(* Visualisation PLC_VISU
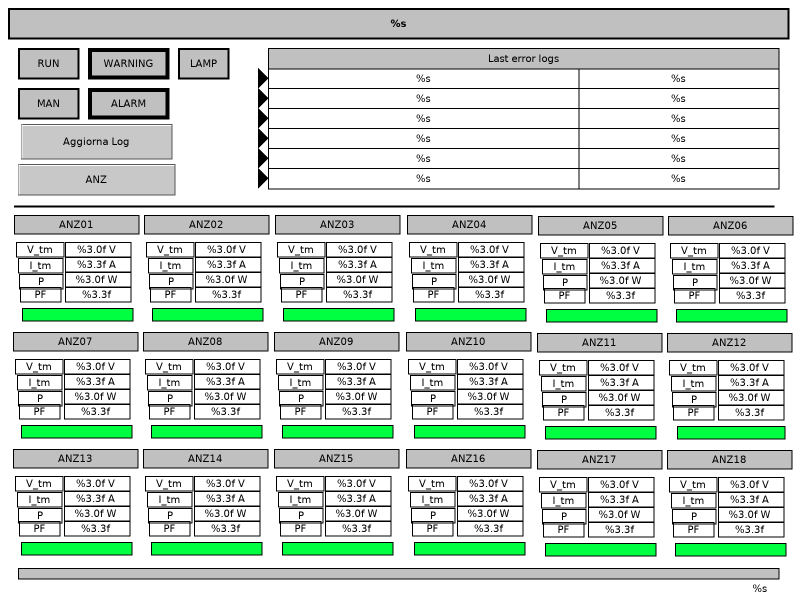
rectangle at (10,10)-(791,41): text "%s"; shows .Plant_NAME
rectangle at (530,580)-(771,601): text "%s"; shows Sys.Time_LogString
rounded rectangle at (20,50)-(81,81): text "RUN"; alarm colour if NOT Mode_Manual; runs INTERN ASSIGN Mode_Manual:=(FALSE)
rounded rectangle at (20,90)-(81,121): text "MAN"; alarm colour if Mode_Manual; runs INTERN ASSIGN Mode_Manual:=(TRUE)
rectangle at (580,70)-(781,91): text "%s"; shows Sys.LastLogs_Msg[0]
polygon at (260,170)-(270,190): invisible if Sys.LastLogs_Idx<>0
rectangle at (580,90)-(781,111): text "%s"; shows Sys.LastLogs_Msg[1]
polygon at (260,70)-(270,90): invisible if Sys.LastLogs_Idx<>1
rectangle at (580,110)-(781,131): text "%s"; shows Sys.LastLogs_Msg[2]
polygon at (260,90)-(270,110): invisible if Sys.LastLogs_Idx<>2
rectangle at (580,130)-(781,151): text "%s"; shows Sys.LastLogs_Msg[3]
polygon at (260,110)-(270,130): invisible if Sys.LastLogs_Idx<>3
rectangle at (580,150)-(781,171): text "%s"; shows Sys.LastLogs_Msg[4]
polygon at (260,130)-(270,150): invisible if Sys.LastLogs_Idx<>4
rectangle at (580,170)-(781,191): text "%s"; shows Sys.LastLogs_Msg[5]
polygon at (260,150)-(270,170): invisible if Sys.LastLogs_Idx<>5
rectangle at (270,70)-(581,91): text "%s"; shows Sys.LastLogs_Dat[0]
rectangle at (270,90)-(581,111): text "%s"; shows Sys.LastLogs_Dat[1]
rectangle at (270,110)-(581,131): text "%s"; shows Sys.LastLogs_Dat[2]
rectangle at (270,130)-(581,151): text "%s"; shows Sys.LastLogs_Dat[3]
rectangle at (270,150)-(581,171): text "%s"; shows Sys.LastLogs_Dat[4]
rectangle at (270,170)-(581,191): text "%s"; shows Sys.LastLogs_Dat[5]
rectangle at (90,90)-(171,121): text "ALARM"; alarm colour if Sys.Alarm; runs INTERN ASSIGN Mode_Manual:=(FALSE)
rectangle at (90,50)-(171,81): text "WARNING"; alarm colour if Sys.Warning; runs INTERN ASSIGN Mode_Manual:=(TRUE)
rectangle at (270,50)-(781,71): text "Last error logs"
rounded rectangle at (180,50)-(231,81): text "LAMP"; alarm colour if LAMP_AL
button at (23,126)-(174,161): text "Aggiorna Log"; taps PLC_PRG.HMI_AggiornaLog
button at (20,166)-(177,197): text "ANZ"; opens VIS_ANZ
rectangle at (67,244)-(133,259): text "%3.0f V"; shows .ANZ01.Voltage_L1_L2
rectangle at (18,244)-(66,259): text "V_tm"
rectangle at (20,260)-(65,275): text "I_tm"
rectangle at (21,276)-(65,291): text "P"
rectangle at (22,289)-(63,304): text "PF"
rectangle at (67,259)-(133,274): text "%3.3f A"; shows .ANZ01.Current_L1
rectangle at (67,274)-(133,289): text "%3.0f W"; shows .ANZ01.ActivePower
rectangle at (67,289)-(133,304): text "%3.3f"; shows .ANZ01.Power_factor_L1
rectangle at (24,310)-(135,323): alarm colour if .ANZ01.AllarmeNodo
rectangle at (16,217)-(141,236): text "ANZ01"
rectangle at (197,244)-(263,259): text "%3.0f V"; shows .ANZ02.Voltage_L1_L2
rectangle at (148,244)-(196,259): text "V_tm"
rectangle at (150,260)-(195,275): text "I_tm"
rectangle at (151,276)-(195,291): text "P"
rectangle at (152,289)-(193,304): text "PF"
rectangle at (197,259)-(263,274): text "%3.3f A"; shows .ANZ02.Current_L1
rectangle at (197,274)-(263,289): text "%3.0f W"; shows .ANZ02.ActivePower
rectangle at (197,289)-(263,304): text "%3.3f"; shows .ANZ02.Power_factor_L1
rectangle at (154,310)-(265,323): alarm colour if .ANZ02.AllarmeNodo
rectangle at (146,217)-(271,236): text "ANZ02"
rectangle at (328,244)-(394,259): text "%3.0f V"; shows .ANZ03.Voltage_L1_L2
rectangle at (279,244)-(327,259): text "V_tm"
rectangle at (281,260)-(326,275): text "I_tm"
rectangle at (282,276)-(326,291): text "P"
rectangle at (283,289)-(324,304): text "PF"
rectangle at (328,259)-(394,274): text "%3.3f A"; shows .ANZ03.Current_L1
rectangle at (328,274)-(394,289): text "%3.0f W"; shows .ANZ03.ActivePower
rectangle at (328,289)-(394,304): text "%3.3f"; shows .ANZ03.Power_factor_L1
rectangle at (285,310)-(396,323): alarm colour if .ANZ03.AllarmeNodo
rectangle at (277,217)-(402,236): text "ANZ03"
rectangle at (460,244)-(526,259): text "%3.0f V"; shows .ANZ04.Voltage_L1_L2
rectangle at (411,244)-(459,259): text "V_tm"
rectangle at (413,260)-(458,275): text "I_tm"
rectangle at (414,276)-(458,291): text "P"
rectangle at (415,289)-(456,304): text "PF"
rectangle at (460,259)-(526,274): text "%3.3f A"; shows .ANZ04.Current_L1
rectangle at (460,274)-(526,289): text "%3.0f W"; shows .ANZ04.ActivePower
rectangle at (460,289)-(526,304): text "%3.3f"; shows .ANZ04.Power_factor_L1
rectangle at (417,310)-(528,323): alarm colour if .ANZ04.AllarmeNodo
rectangle at (409,217)-(534,236): text "ANZ04"
rectangle at (591,245)-(657,260): text "%3.0f V"; shows .ANZ05.Voltage_L1_L2
rectangle at (542,245)-(590,260): text "V_tm"
rectangle at (544,261)-(589,276): text "I_tm"
rectangle at (545,277)-(589,292): text "P"
rectangle at (546,290)-(587,305): text "PF"
rectangle at (591,260)-(657,275): text "%3.3f A"; shows .ANZ05.Current_L1
rectangle at (591,275)-(657,290): text "%3.0f W"; shows .ANZ05.ActivePower
rectangle at (591,290)-(657,305): text "%3.3f"; shows .ANZ05.Power_factor_L1
rectangle at (548,311)-(659,324): alarm colour if .ANZ05.AllarmeNodo
rectangle at (540,218)-(665,237): text "ANZ05"
rectangle at (721,245)-(787,260): text "%3.0f V"; shows .ANZ06.Voltage_L1_L2
rectangle at (672,245)-(720,260): text "V_tm"
rectangle at (674,261)-(719,276): text "I_tm"
rectangle at (675,277)-(719,292): text "P"
rectangle at (676,290)-(717,305): text "PF"
rectangle at (721,260)-(787,275): text "%3.3f A"; shows .ANZ06.Current_L1
rectangle at (721,275)-(787,290): text "%3.0f W"; shows .ANZ06.ActivePower
rectangle at (721,290)-(787,305): text "%3.3f"; shows .ANZ06.Power_factor_L1
rectangle at (678,311)-(789,324): alarm colour if .ANZ06.AllarmeNodo
rectangle at (670,218)-(795,237): text "ANZ06"
rectangle at (66,361)-(132,376): text "%3.0f V"; shows .ANZ07.Voltage_L1_L2
rectangle at (17,361)-(65,376): text "V_tm"
rectangle at (19,377)-(64,392): text "I_tm"
rectangle at (20,393)-(64,408): text "P"
rectangle at (21,406)-(62,421): text "PF"
rectangle at (66,376)-(132,391): text "%3.3f A"; shows .ANZ07.Current_L1
rectangle at (66,391)-(132,406): text "%3.0f W"; shows .ANZ07.ActivePower
rectangle at (66,406)-(132,421): text "%3.3f"; shows .ANZ07.Power_factor_L1
rectangle at (23,427)-(134,440): alarm colour if .ANZ07.AllarmeNodo
rectangle at (15,334)-(140,353): text "ANZ07"
rectangle at (196,361)-(262,376): text "%3.0f V"; shows .ANZ08.Voltage_L1_L2
rectangle at (147,361)-(195,376): text "V_tm"
rectangle at (149,377)-(194,392): text "I_tm"
rectangle at (150,393)-(194,408): text "P"
rectangle at (151,406)-(192,421): text "PF"
rectangle at (196,376)-(262,391): text "%3.3f A"; shows .ANZ08.Current_L1
rectangle at (196,391)-(262,406): text "%3.0f W"; shows .ANZ08.ActivePower
rectangle at (196,406)-(262,421): text "%3.3f"; shows .ANZ08.Power_factor_L1
rectangle at (153,427)-(264,440): alarm colour if .ANZ08.AllarmeNodo
rectangle at (145,334)-(270,353): text "ANZ08"
rectangle at (327,361)-(393,376): text "%3.0f V"; shows .ANZ09.Voltage_L1_L2
rectangle at (278,361)-(326,376): text "V_tm"
rectangle at (280,377)-(325,392): text "I_tm"
rectangle at (281,393)-(325,408): text "P"
rectangle at (282,406)-(323,421): text "PF"
rectangle at (327,376)-(393,391): text "%3.3f A"; shows .ANZ09.Current_L1
rectangle at (327,391)-(393,406): text "%3.0f W"; shows .ANZ09.ActivePower
rectangle at (327,406)-(393,421): text "%3.3f"; shows .ANZ09.Power_factor_L1
rectangle at (284,427)-(395,440): alarm colour if .ANZ09.AllarmeNodo
rectangle at (276,334)-(401,353): text "ANZ09"
rectangle at (459,361)-(525,376): text "%3.0f V"; shows .ANZ10.Voltage_L1_L2
rectangle at (410,361)-(458,376): text "V_tm"
rectangle at (412,377)-(457,392): text "I_tm"
rectangle at (413,393)-(457,408): text "P"
rectangle at (414,406)-(455,421): text "PF"
rectangle at (459,376)-(525,391): text "%3.3f A"; shows .ANZ10.Current_L1
rectangle at (459,391)-(525,406): text "%3.0f W"; shows .ANZ10.ActivePower
rectangle at (459,406)-(525,421): text "%3.3f"; shows .ANZ10.Power_factor_L1
rectangle at (416,427)-(527,440): alarm colour if .ANZ10.AllarmeNodo
rectangle at (408,334)-(533,353): text "ANZ10"
rectangle at (590,362)-(656,377): text "%3.0f V"; shows .ANZ11.Voltage_L1_L2
rectangle at (541,362)-(589,377): text "V_tm"
rectangle at (543,378)-(588,393): text "I_tm"
rectangle at (544,394)-(588,409): text "P"
rectangle at (545,407)-(586,422): text "PF"
rectangle at (590,377)-(656,392): text "%3.3f A"; shows .ANZ11.Current_L1
rectangle at (590,392)-(656,407): text "%3.0f W"; shows .ANZ11.ActivePower
rectangle at (590,407)-(656,422): text "%3.3f"; shows .ANZ11.Power_factor_L1
rectangle at (547,428)-(658,441): alarm colour if .ANZ11.AllarmeNodo
rectangle at (539,335)-(664,354): text "ANZ11"
rectangle at (720,362)-(786,377): text "%3.0f V"; shows .ANZ12.Voltage_L1_L2
rectangle at (671,362)-(719,377): text "V_tm"
rectangle at (673,378)-(718,393): text "I_tm"
rectangle at (674,394)-(718,409): text "P"
rectangle at (675,407)-(716,422): text "PF"
rectangle at (720,377)-(786,392): text "%3.3f A"; shows .ANZ12.Current_L1
rectangle at (720,392)-(786,407): text "%3.0f W"; shows .ANZ12.ActivePower
rectangle at (720,407)-(786,422): text "%3.3f"; shows .ANZ12.Power_factor_L1
rectangle at (669,335)-(794,354): text "ANZ12"
rectangle at (66,478)-(132,493): text "%3.0f V"; shows .ANZ13.Voltage_L1_L2
rectangle at (17,478)-(65,493): text "V_tm"
rectangle at (19,494)-(64,509): text "I_tm"
rectangle at (20,510)-(64,525): text "P"
rectangle at (21,523)-(62,538): text "PF"
rectangle at (66,493)-(132,508): text "%3.3f A"; shows .ANZ13.Current_L1
rectangle at (66,508)-(132,523): text "%3.0f W"; shows .ANZ13.ActivePower
rectangle at (66,523)-(132,538): text "%3.3f"; shows .ANZ13.Power_factor_L1
rectangle at (23,544)-(134,557): alarm colour if .ANZ13.AllarmeNodo
rectangle at (15,451)-(140,470): text "ANZ13"
rectangle at (196,478)-(262,493): text "%3.0f V"; shows .ANZ14.Voltage_L1_L2
rectangle at (147,478)-(195,493): text "V_tm"
rectangle at (149,494)-(194,509): text "I_tm"
rectangle at (150,510)-(194,525): text "P"
rectangle at (151,523)-(192,538): text "PF"
rectangle at (196,493)-(262,508): text "%3.3f A"; shows .ANZ14.Current_L1
rectangle at (196,508)-(262,523): text "%3.0f W"; shows .ANZ14.ActivePower
rectangle at (196,523)-(262,538): text "%3.3f"; shows .ANZ14.Power_factor_L1
rectangle at (153,544)-(264,557): alarm colour if .ANZ14.AllarmeNodo
rectangle at (145,451)-(270,470): text "ANZ14"
rectangle at (327,478)-(393,493): text "%3.0f V"; shows .ANZ15.Voltage_L1_L2
rectangle at (278,478)-(326,493): text "V_tm"
rectangle at (280,494)-(325,509): text "I_tm"
rectangle at (281,510)-(325,525): text "P"
rectangle at (282,523)-(323,538): text "PF"
rectangle at (327,493)-(393,508): text "%3.3f A"; shows .ANZ15.Current_L1
rectangle at (327,508)-(393,523): text "%3.0f W"; shows .ANZ15.ActivePower
rectangle at (327,523)-(393,538): text "%3.3f"; shows .ANZ15.Power_factor_L1
rectangle at (284,544)-(395,557): alarm colour if .ANZ15.AllarmeNodo
rectangle at (276,451)-(401,470): text "ANZ15"
rectangle at (459,478)-(525,493): text "%3.0f V"; shows .ANZ16.Voltage_L1_L2
rectangle at (410,478)-(458,493): text "V_tm"
rectangle at (412,494)-(457,509): text "I_tm"
rectangle at (413,510)-(457,525): text "P"
rectangle at (414,523)-(455,538): text "PF"
rectangle at (459,493)-(525,508): text "%3.3f A"; shows .ANZ16.Current_L1
rectangle at (459,508)-(525,523): text "%3.0f W"; shows .ANZ16.ActivePower
rectangle at (459,523)-(525,538): text "%3.3f"; shows .ANZ16.Power_factor_L1
rectangle at (416,544)-(527,557): alarm colour if .ANZ16.AllarmeNodo
rectangle at (408,451)-(533,470): text "ANZ16"
rectangle at (590,479)-(656,494): text "%3.0f V"; shows .ANZ17.Voltage_L1_L2
rectangle at (541,479)-(589,494): text "V_tm"
rectangle at (543,495)-(588,510): text "I_tm"
rectangle at (544,511)-(588,526): text "P"
rectangle at (545,524)-(586,539): text "PF"
rectangle at (590,494)-(656,509): text "%3.3f A"; shows .ANZ17.Current_L1
rectangle at (590,509)-(656,524): text "%3.0f W"; shows .ANZ17.ActivePower
rectangle at (590,524)-(656,539): text "%3.3f"; shows .ANZ17.Power_factor_L1
rectangle at (547,545)-(658,558): alarm colour if .ANZ17.AllarmeNodo
rectangle at (539,452)-(664,471): text "ANZ17"
rectangle at (720,479)-(786,494): text "%3.0f V"; shows .ANZ18.Voltage_L1_L2
rectangle at (671,479)-(719,494): text "V_tm"
rectangle at (673,495)-(718,510): text "I_tm"
rectangle at (674,511)-(718,526): text "P"
rectangle at (675,524)-(716,539): text "PF"
rectangle at (720,494)-(786,509): text "%3.3f A"; shows .ANZ18.Current_L1
rectangle at (720,509)-(786,524): text "%3.0f W"; shows .ANZ18.ActivePower
rectangle at (720,524)-(786,539): text "%3.3f"; shows .ANZ18.Power_factor_L1
rectangle at (677,545)-(788,558): alarm colour if .ANZ18.AllarmeNodo
rectangle at (669,452)-(794,471): text "ANZ18"
rectangle at (679,428)-(787,441): alarm colour if .ANZ12.AllarmeNodo
20 more shapes without text or variables
*)

(* Visualisation VIS_ANZ
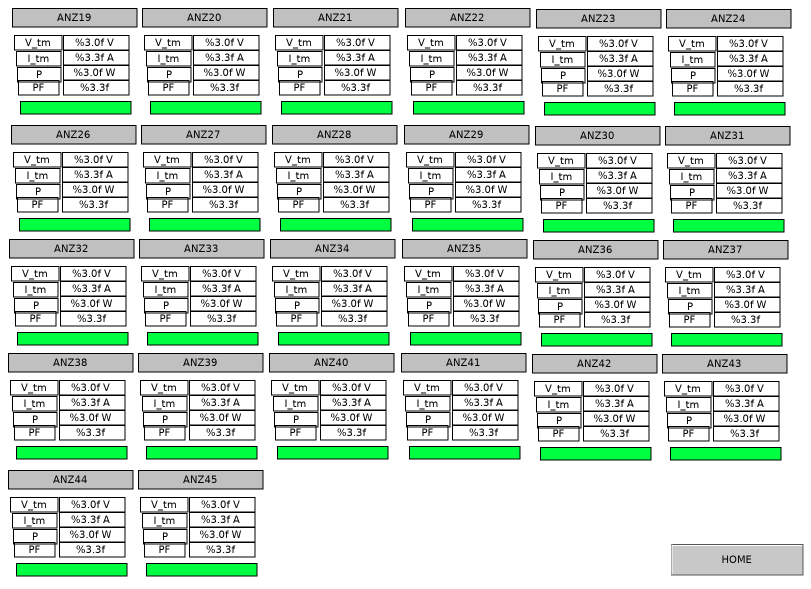
rectangle at (51,38)-(117,53): text "%3.0f V"; shows .ANZ19.Voltage_L1_L2
rectangle at (2,38)-(50,53): text "V_tm"
rectangle at (4,54)-(49,69): text "I_tm"
rectangle at (5,70)-(49,85): text "P"
rectangle at (6,83)-(47,98): text "PF"
rectangle at (51,53)-(117,68): text "%3.3f A"; shows .ANZ19.Current_L1
rectangle at (51,68)-(117,83): text "%3.0f W"; shows .ANZ19.ActivePower
rectangle at (51,83)-(117,98): text "%3.3f"; shows .ANZ19.Power_factor_L1
rectangle at (8,104)-(119,117): alarm colour if .ANZ19.AllarmeNodo
rectangle at (0,11)-(125,30): text "ANZ19"
rectangle at (181,38)-(247,53): text "%3.0f V"; shows .ANZ20.Voltage_L1_L2
rectangle at (132,38)-(180,53): text "V_tm"
rectangle at (134,54)-(179,69): text "I_tm"
rectangle at (135,70)-(179,85): text "P"
rectangle at (136,83)-(177,98): text "PF"
rectangle at (181,53)-(247,68): text "%3.3f A"; shows .ANZ20.Current_L1
rectangle at (181,68)-(247,83): text "%3.0f W"; shows .ANZ20.ActivePower
rectangle at (181,83)-(247,98): text "%3.3f"; shows .ANZ20.Power_factor_L1
rectangle at (138,104)-(249,117): alarm colour if .ANZ20.AllarmeNodo
rectangle at (130,11)-(255,30): text "ANZ20"
rectangle at (312,38)-(378,53): text "%3.0f V"; shows .ANZ21.Voltage_L1_L2
rectangle at (263,38)-(311,53): text "V_tm"
rectangle at (265,54)-(310,69): text "I_tm"
rectangle at (266,70)-(310,85): text "P"
rectangle at (267,83)-(308,98): text "PF"
rectangle at (312,53)-(378,68): text "%3.3f A"; shows .ANZ21.Current_L1
rectangle at (312,68)-(378,83): text "%3.0f W"; shows .ANZ21.ActivePower
rectangle at (312,83)-(378,98): text "%3.3f"; shows .ANZ21.Power_factor_L1
rectangle at (269,104)-(380,117): alarm colour if .ANZ21.AllarmeNodo
rectangle at (261,11)-(386,30): text "ANZ21"
rectangle at (444,38)-(510,53): text "%3.0f V"; shows .ANZ22.Voltage_L1_L2
rectangle at (395,38)-(443,53): text "V_tm"
rectangle at (397,54)-(442,69): text "I_tm"
rectangle at (398,70)-(442,85): text "P"
rectangle at (399,83)-(440,98): text "PF"
rectangle at (444,53)-(510,68): text "%3.3f A"; shows .ANZ22.Current_L1
rectangle at (444,68)-(510,83): text "%3.0f W"; shows .ANZ22.ActivePower
rectangle at (444,83)-(510,98): text "%3.3f"; shows .ANZ22.Power_factor_L1
rectangle at (401,104)-(512,117): alarm colour if .ANZ22.AllarmeNodo
rectangle at (393,11)-(518,30): text "ANZ22"
rectangle at (575,39)-(641,54): text "%3.0f V"; shows .ANZ23.Voltage_L1_L2
rectangle at (526,39)-(574,54): text "V_tm"
rectangle at (528,55)-(573,70): text "I_tm"
rectangle at (529,71)-(573,86): text "P"
rectangle at (530,84)-(571,99): text "PF"
rectangle at (575,54)-(641,69): text "%3.3f A"; shows .ANZ23.Current_L1
rectangle at (575,69)-(641,84): text "%3.0f W"; shows .ANZ23.ActivePower
rectangle at (575,84)-(641,99): text "%3.3f"; shows .ANZ23.Power_factor_L1
rectangle at (532,105)-(643,118): alarm colour if .ANZ23.AllarmeNodo
rectangle at (524,12)-(649,31): text "ANZ23"
rectangle at (705,39)-(771,54): text "%3.0f V"; shows .ANZ24.Voltage_L1_L2
rectangle at (656,39)-(704,54): text "V_tm"
rectangle at (658,55)-(703,70): text "I_tm"
rectangle at (659,71)-(703,86): text "P"
rectangle at (660,84)-(701,99): text "PF"
rectangle at (705,54)-(771,69): text "%3.3f A"; shows .ANZ24.Current_L1
rectangle at (705,69)-(771,84): text "%3.0f W"; shows .ANZ24.ActivePower
rectangle at (705,84)-(771,99): text "%3.3f"; shows .ANZ24.Power_factor_L1
rectangle at (662,105)-(773,118): alarm colour if .ANZ24.AllarmeNodo
rectangle at (654,12)-(779,31): text "ANZ24"
rectangle at (50,155)-(116,170): text "%3.0f V"; shows .ANZ26.Voltage_L1_L2
rectangle at (1,155)-(49,170): text "V_tm"
rectangle at (3,171)-(48,186): text "I_tm"
rectangle at (4,187)-(48,202): text "P"
rectangle at (5,200)-(46,215): text "PF"
rectangle at (50,170)-(116,185): text "%3.3f A"; shows .ANZ26.Current_L1
rectangle at (50,185)-(116,200): text "%3.0f W"; shows .ANZ26.ActivePower
rectangle at (50,200)-(116,215): text "%3.3f"; shows .ANZ26.Power_factor_L1
rectangle at (7,221)-(118,234): alarm colour if .ANZ26.AllarmeNodo
rectangle at (-1,128)-(124,147): text "ANZ26"
rectangle at (180,155)-(246,170): text "%3.0f V"; shows .ANZ27.Voltage_L1_L2
rectangle at (131,155)-(179,170): text "V_tm"
rectangle at (133,171)-(178,186): text "I_tm"
rectangle at (134,187)-(178,202): text "P"
rectangle at (135,200)-(176,215): text "PF"
rectangle at (180,170)-(246,185): text "%3.3f A"; shows .ANZ27.Current_L1
rectangle at (180,185)-(246,200): text "%3.0f W"; shows .ANZ27.ActivePower
rectangle at (180,200)-(246,215): text "%3.3f"; shows .ANZ27.Power_factor_L1
rectangle at (137,221)-(248,234): alarm colour if .ANZ27.AllarmeNodo
rectangle at (129,128)-(254,147): text "ANZ27"
rectangle at (311,155)-(377,170): text "%3.0f V"; shows .ANZ28.Voltage_L1_L2
rectangle at (262,155)-(310,170): text "V_tm"
rectangle at (264,171)-(309,186): text "I_tm"
rectangle at (265,187)-(309,202): text "P"
rectangle at (266,200)-(307,215): text "PF"
rectangle at (311,170)-(377,185): text "%3.3f A"; shows .ANZ28.Current_L1
rectangle at (311,185)-(377,200): text "%3.0f W"; shows .ANZ28.ActivePower
rectangle at (311,200)-(377,215): text "%3.3f"; shows .ANZ28.Power_factor_L1
rectangle at (268,221)-(379,234): alarm colour if .ANZ28.AllarmeNodo
rectangle at (260,128)-(385,147): text "ANZ28"
rectangle at (443,155)-(509,170): text "%3.0f V"; shows .ANZ29.Voltage_L1_L2
rectangle at (394,155)-(442,170): text "V_tm"
rectangle at (396,171)-(441,186): text "I_tm"
rectangle at (397,187)-(441,202): text "P"
rectangle at (398,200)-(439,215): text "PF"
rectangle at (443,170)-(509,185): text "%3.3f A"; shows .ANZ29.Current_L1
rectangle at (443,185)-(509,200): text "%3.0f W"; shows .ANZ29.ActivePower
rectangle at (443,200)-(509,215): text "%3.3f"; shows .ANZ29.Power_factor_L1
rectangle at (400,221)-(511,234): alarm colour if .ANZ29.AllarmeNodo
rectangle at (392,128)-(517,147): text "ANZ29"
rectangle at (574,156)-(640,171): text "%3.0f V"; shows .ANZ30.Voltage_L1_L2
rectangle at (525,156)-(573,171): text "V_tm"
rectangle at (527,172)-(572,187): text "I_tm"
rectangle at (528,188)-(572,203): text "P"
rectangle at (529,201)-(570,216): text "PF"
rectangle at (574,171)-(640,186): text "%3.3f A"; shows .ANZ30.Current_L1
rectangle at (574,186)-(640,201): text "%3.0f W"; shows .ANZ30.ActivePower
rectangle at (574,201)-(640,216): text "%3.3f"; shows .ANZ30.Power_factor_L1
rectangle at (531,222)-(642,235): alarm colour if .ANZ30.AllarmeNodo
rectangle at (523,129)-(648,148): text "ANZ30"
rectangle at (704,156)-(770,171): text "%3.0f V"; shows .ANZ31.Voltage_L1_L2
rectangle at (655,156)-(703,171): text "V_tm"
rectangle at (657,172)-(702,187): text "I_tm"
rectangle at (658,188)-(702,203): text "P"
rectangle at (659,201)-(700,216): text "PF"
rectangle at (704,171)-(770,186): text "%3.3f A"; shows .ANZ31.Current_L1
rectangle at (704,186)-(770,201): text "%3.0f W"; shows .ANZ31.ActivePower
rectangle at (704,201)-(770,216): text "%3.3f"; shows .ANZ31.Power_factor_L1
rectangle at (661,222)-(772,235): alarm colour if .ANZ31.AllarmeNodo
rectangle at (653,129)-(778,148): text "ANZ31"
rectangle at (48,269)-(114,284): text "%3.0f V"; shows .ANZ32.Voltage_L1_L2
rectangle at (-1,269)-(47,284): text "V_tm"
rectangle at (1,285)-(46,300): text "I_tm"
rectangle at (2,301)-(46,316): text "P"
rectangle at (3,314)-(44,329): text "PF"
rectangle at (48,284)-(114,299): text "%3.3f A"; shows .ANZ32.Current_L1
rectangle at (48,299)-(114,314): text "%3.0f W"; shows .ANZ32.ActivePower
rectangle at (48,314)-(114,329): text "%3.3f"; shows .ANZ32.Power_factor_L1
rectangle at (5,335)-(116,348): alarm colour if .ANZ32.AllarmeNodo
rectangle at (-3,242)-(122,261): text "ANZ32"
rectangle at (178,269)-(244,284): text "%3.0f V"; shows .ANZ33.Voltage_L1_L2
rectangle at (129,269)-(177,284): text "V_tm"
rectangle at (131,285)-(176,300): text "I_tm"
rectangle at (132,301)-(176,316): text "P"
rectangle at (133,314)-(174,329): text "PF"
rectangle at (178,284)-(244,299): text "%3.3f A"; shows .ANZ33.Current_L1
rectangle at (178,299)-(244,314): text "%3.0f W"; shows .ANZ33.ActivePower
rectangle at (178,314)-(244,329): text "%3.3f"; shows .ANZ33.Power_factor_L1
rectangle at (135,335)-(246,348): alarm colour if .ANZ33.AllarmeNodo
rectangle at (127,242)-(252,261): text "ANZ33"
rectangle at (309,269)-(375,284): text "%3.0f V"; shows .ANZ34.Voltage_L1_L2
rectangle at (260,269)-(308,284): text "V_tm"
rectangle at (262,285)-(307,300): text "I_tm"
rectangle at (263,301)-(307,316): text "P"
rectangle at (264,314)-(305,329): text "PF"
rectangle at (309,284)-(375,299): text "%3.3f A"; shows .ANZ34.Current_L1
rectangle at (309,299)-(375,314): text "%3.0f W"; shows .ANZ34.ActivePower
rectangle at (309,314)-(375,329): text "%3.3f"; shows .ANZ34.Power_factor_L1
rectangle at (266,335)-(377,348): alarm colour if .ANZ34.AllarmeNodo
rectangle at (258,242)-(383,261): text "ANZ34"
rectangle at (441,269)-(507,284): text "%3.0f V"; shows .ANZ35.Voltage_L1_L2
rectangle at (392,269)-(440,284): text "V_tm"
rectangle at (394,285)-(439,300): text "I_tm"
rectangle at (395,301)-(439,316): text "P"
rectangle at (396,314)-(437,329): text "PF"
rectangle at (441,284)-(507,299): text "%3.3f A"; shows .ANZ35.Current_L1
rectangle at (441,299)-(507,314): text "%3.0f W"; shows .ANZ35.ActivePower
rectangle at (441,314)-(507,329): text "%3.3f"; shows .ANZ35.Power_factor_L1
rectangle at (398,335)-(509,348): alarm colour if .ANZ35.AllarmeNodo
rectangle at (390,242)-(515,261): text "ANZ35"
rectangle at (572,270)-(638,285): text "%3.0f V"; shows .ANZ36.Voltage_L1_L2
rectangle at (523,270)-(571,285): text "V_tm"
rectangle at (525,286)-(570,301): text "I_tm"
rectangle at (526,302)-(570,317): text "P"
rectangle at (527,315)-(568,330): text "PF"
rectangle at (572,285)-(638,300): text "%3.3f A"; shows .ANZ36.Current_L1
rectangle at (572,300)-(638,315): text "%3.0f W"; shows .ANZ36.ActivePower
rectangle at (572,315)-(638,330): text "%3.3f"; shows .ANZ36.Power_factor_L1
rectangle at (529,336)-(640,349): alarm colour if .ANZ36.AllarmeNodo
rectangle at (521,243)-(646,262): text "ANZ36"
rectangle at (702,270)-(768,285): text "%3.0f V"; shows .ANZ37.Voltage_L1_L2
rectangle at (653,270)-(701,285): text "V_tm"
rectangle at (655,286)-(700,301): text "I_tm"
rectangle at (656,302)-(700,317): text "P"
rectangle at (657,315)-(698,330): text "PF"
rectangle at (702,285)-(768,300): text "%3.3f A"; shows .ANZ37.Current_L1
rectangle at (702,300)-(768,315): text "%3.0f W"; shows .ANZ37.ActivePower
rectangle at (702,315)-(768,330): text "%3.3f"; shows .ANZ37.Power_factor_L1
rectangle at (659,336)-(770,349): alarm colour if .ANZ37.AllarmeNodo
rectangle at (651,243)-(776,262): text "ANZ37"
rectangle at (47,383)-(113,398): text "%3.0f V"; shows .ANZ38.Voltage_L1_L2
rectangle at (-2,383)-(46,398): text "V_tm"
rectangle at (0,399)-(45,414): text "I_tm"
rectangle at (1,415)-(45,430): text "P"
rectangle at (2,428)-(43,443): text "PF"
rectangle at (47,398)-(113,413): text "%3.3f A"; shows .ANZ38.Current_L1
rectangle at (47,413)-(113,428): text "%3.0f W"; shows .ANZ38.ActivePower
rectangle at (47,428)-(113,443): text "%3.3f"; shows .ANZ38.Power_factor_L1
rectangle at (4,449)-(115,462): alarm colour if .ANZ38.AllarmeNodo
rectangle at (-4,356)-(121,375): text "ANZ38"
rectangle at (177,383)-(243,398): text "%3.0f V"; shows .ANZ39.Voltage_L1_L2
rectangle at (128,383)-(176,398): text "V_tm"
rectangle at (130,399)-(175,414): text "I_tm"
rectangle at (131,415)-(175,430): text "P"
rectangle at (132,428)-(173,443): text "PF"
rectangle at (177,398)-(243,413): text "%3.3f A"; shows .ANZ39.Current_L1
rectangle at (177,413)-(243,428): text "%3.0f W"; shows .ANZ39.ActivePower
rectangle at (177,428)-(243,443): text "%3.3f"; shows .ANZ39.Power_factor_L1
rectangle at (134,449)-(245,462): alarm colour if .ANZ39.AllarmeNodo
rectangle at (126,356)-(251,375): text "ANZ39"
rectangle at (308,383)-(374,398): text "%3.0f V"; shows .ANZ40.Voltage_L1_L2
rectangle at (259,383)-(307,398): text "V_tm"
rectangle at (261,399)-(306,414): text "I_tm"
rectangle at (262,415)-(306,430): text "P"
rectangle at (263,428)-(304,443): text "PF"
rectangle at (308,398)-(374,413): text "%3.3f A"; shows .ANZ40.Current_L1
rectangle at (308,413)-(374,428): text "%3.0f W"; shows .ANZ40.ActivePower
rectangle at (308,428)-(374,443): text "%3.3f"; shows .ANZ40.Power_factor_L1
rectangle at (265,449)-(376,462): alarm colour if .ANZ40.AllarmeNodo
rectangle at (257,356)-(382,375): text "ANZ40"
rectangle at (440,383)-(506,398): text "%3.0f V"; shows .ANZ41.Voltage_L1_L2
rectangle at (391,383)-(439,398): text "V_tm"
rectangle at (393,399)-(438,414): text "I_tm"
rectangle at (394,415)-(438,430): text "P"
rectangle at (395,428)-(436,443): text "PF"
rectangle at (440,398)-(506,413): text "%3.3f A"; shows .ANZ41.Current_L1
rectangle at (440,413)-(506,428): text "%3.0f W"; shows .ANZ41.ActivePower
rectangle at (440,428)-(506,443): text "%3.3f"; shows .ANZ41.Power_factor_L1
rectangle at (397,449)-(508,462): alarm colour if .ANZ41.AllarmeNodo
rectangle at (389,356)-(514,375): text "ANZ41"
rectangle at (571,384)-(637,399): text "%3.0f V"; shows .ANZ42.Voltage_L1_L2
rectangle at (522,384)-(570,399): text "V_tm"
rectangle at (524,400)-(569,415): text "I_tm"
rectangle at (525,416)-(569,431): text "P"
rectangle at (526,429)-(567,444): text "PF"
rectangle at (571,399)-(637,414): text "%3.3f A"; shows .ANZ42.Current_L1
rectangle at (571,414)-(637,429): text "%3.0f W"; shows .ANZ42.ActivePower
rectangle at (571,429)-(637,444): text "%3.3f"; shows .ANZ42.Power_factor_L1
rectangle at (528,450)-(639,463): alarm colour if .ANZ42.AllarmeNodo
rectangle at (520,357)-(645,376): text "ANZ42"
rectangle at (701,384)-(767,399): text "%3.0f V"; shows .ANZ43.Voltage_L1_L2
rectangle at (652,384)-(700,399): text "V_tm"
rectangle at (654,400)-(699,415): text "I_tm"
rectangle at (655,416)-(699,431): text "P"
rectangle at (656,429)-(697,444): text "PF"
rectangle at (701,399)-(767,414): text "%3.3f A"; shows .ANZ43.Current_L1
rectangle at (701,414)-(767,429): text "%3.0f W"; shows .ANZ43.ActivePower
rectangle at (701,429)-(767,444): text "%3.3f"; shows .ANZ43.Power_factor_L1
rectangle at (658,450)-(769,463): alarm colour if .ANZ43.AllarmeNodo
rectangle at (650,357)-(775,376): text "ANZ43"
rectangle at (47,500)-(113,515): text "%3.0f V"; shows .ANZ44.Voltage_L1_L2
rectangle at (-2,500)-(46,515): text "V_tm"
rectangle at (0,516)-(45,531): text "I_tm"
rectangle at (1,532)-(45,547): text "P"
rectangle at (2,545)-(43,560): text "PF"
rectangle at (47,515)-(113,530): text "%3.3f A"; shows .ANZ44.Current_L1
rectangle at (47,530)-(113,545): text "%3.0f W"; shows .ANZ44.ActivePower
rectangle at (47,545)-(113,560): text "%3.3f"; shows .ANZ44.Power_factor_L1
rectangle at (4,566)-(115,579): alarm colour if .ANZ44.AllarmeNodo
rectangle at (-4,473)-(121,492): text "ANZ44"
rectangle at (177,500)-(243,515): text "%3.0f V"; shows .ANZ45.Voltage_L1_L2
rectangle at (128,500)-(176,515): text "V_tm"
rectangle at (130,516)-(175,531): text "I_tm"
rectangle at (131,532)-(175,547): text "P"
rectangle at (132,545)-(173,560): text "PF"
rectangle at (177,515)-(243,530): text "%3.3f A"; shows .ANZ45.Current_L1
rectangle at (177,530)-(243,545): text "%3.0f W"; shows .ANZ45.ActivePower
rectangle at (177,545)-(243,560): text "%3.3f"; shows .ANZ45.Power_factor_L1
rectangle at (134,566)-(245,579): alarm colour if .ANZ45.AllarmeNodo
rectangle at (126,473)-(251,492): text "ANZ45"
button at (659,547)-(791,578): text "HOME"; opens PLC_VISU
26 more shapes without text or variables
*)
